Staubli VAL3: Vplus.dtx

jointRx jApproBox = {j4=-92.220275879, j3=-91.7603, j5=93.350395203, j1=-156.02204895, j2=-0.296387, j6=-204.139266968
}
jointRx jApproCam = {j4=-180, j3=-82.2022, j5=103.994537354, j1=17.642303467, j2=3.86292, j6=-29.504484177}
jointRx jApproConveyor = {j4=-180.000076294, j3=-104.09, j5=92.340240479, j1=-158.040847778, j2=16.4304, j6=-180.000152588}
jointRx jApproImm = {j4=-185.301483154, j3=-141.503, j5=-47.082424164, j1=105.804260254, j2=4.10028, j6=197.839569092}
jointRx jApproInspect = {j4=-180.122924805, j3=-94.165, j5=107.282814026, j1=79.97895813, j2=19.1074, j6=-27.049661636}
jointRx jApproReject = {j4=-180.000076294, j3=-82.9248, j5=105.547271729, j1=-36.019268036, j2=7.53623, j6=-53.689052582}
jointRx jApproSink = {j4=-180, j3=-82.9248, j5=105.547271729, j1=57.782627106, j2=7.53623, j6=-53.689052582}
jointRx jApproTurn = {j4=-180.000076294, j3=-91.6509, j5=105.937507629, j1=-68.973823547, j2=15.2445, j6=-24.155277252}
jointRx jApproWeld = {j4=-180, j3=-97.4879, j5=76.231643677, j1=-117.552749634, j2=-9.04277, j6=-203.299514771}
pointRx pCamCoords = {rx=0, x=143.13, ry=0, z=0, rz=-124.14, y=76.87, fatherId=world[0]}
pointRx pCamOrig = {rx=0.088055, x=-777.298, ry=177.401, z=14.3041, rz=-179.442, y=67.5964, fatherId=world[0]}
pointRx pCamX = {rx=0.0877556, x=-688.671, ry=177.399, z=15.1582, rz=-179.444, y=-158.575, fatherId=world[0]}
pointRx pCamY = {rx=0.0885309, x=-610.055, ry=177.399, z=12.4062, rz=-179.445, y=133.542, fatherId=world[0]}
tool pGripper0deg = {rx=0, x=0, ry=0, z=400, rz=0, ioLink=valve1, y=2, fatherId=flange[0]}
tool pGripper90deg = {rx=-89.9802, x=0, ry=0, z=312.5, rz=0, ioLink=valve1, y=-87.5, fatherId=flange[0]}
jointRx jHome = {j4=-180, j3=-104.09, j5=92.340240479, j1=-89.999916077, j2=16.4304, j6=-180.000152588}
pointRx pInspection = {rx=-0.828271, x=-402.297, ry=179.533, z=45.3187, rz=71.0887, y=-398.404, fatherId=world[0]}
pointRx pPickImm = {rx=-0.0335721, x=713.865, ry=88.1187, z=-110.012, rz=142.138, y=-1042.29, fatherId=world[0]}
pointRx pPickLoc = {rx=-0.45978, x=-648.514, ry=-179.559, z=13.9554, rz=-173.639, y=-37.8477, fatherId=world[0]}
pointRx pPickTurn = {rx=0.649757, x=-388.63, ry=179.139, z=10.1432, rz=-89.9458, y=350.625, fatherId=world[0]}
pointRx pPickWeld = {rx=-0.721699, x=-100.432, ry=-2.56053, z=-8.67817, rz=-71.824, y=700.057, fatherId=world[0]}
pointRx pPlaceBox[3]
  [0] = {rx=-0.00931083, x=744.888, ry=26.8991, z=177.661, rz=31.4855, y=890.517, fatherId=world[0]}
  [1] = {rx=-0.00931083, x=744.888, ry=26.8991, z=177.661, rz=31.4855, y=890.517, fatherId=world[0]}
  [2] = {rx=-0.00931083, x=744.888, ry=26.8991, z=177.661, rz=31.4855, y=890.517, fatherId=world[0]}
  [3] = {rx=-0.00931083, x=744.888, ry=26.8991, z=177.661, rz=31.4855, y=890.517, fatherId=world[0]}
pointRx pPlaceBoxRejec = {rx=-33.9923, x=393.165, ry=-30.0331, z=496.328, rz=22.9459, y=839.667, fatherId=world[0]}
pointRx pPlaceCover
  [0] = {rx=-3.39884, x=-140.67, ry=-2.89406, z=11.5788, rz=-72.075, y=727.524, fatherId=world[0]}
  [1] = {rx=4.46172, x=-55.7643, ry=-2.8981, z=-7.34839, rz=-72.4729, y=700.328, fatherId=world[0]}
pointRx pPlaceImm = {rx=2.40564, x=695.557, ry=88.1161, z=-100.844, rz=140.773, y=-867.761, fatherId=world[0]}
pointRx pPlaceReject = {rx=-0.758349, x=-362.79, ry=179.442, z=-135.753, rz=-101.683, y=177.761, fatherId=world[0]}
pointRx pPlaceSink = {rx=23.517, x=-427.516, ry=179.533, z=57.5011, rz=68.2962, y=-256.819, fatherId=world[0]}
pointRx pPlaceTurn = {rx=-2.72726, x=-533.365, ry=-4.55086, z=274.72, rz=-93.0403, y=527.16, fatherId=world[0]}
pointRx pPlaceWeld = {rx=-0.773504, x=38.7997, ry=178.381, z=-171.963, rz=108.632, y=668.081, fatherId=world[0]}
pointRx pPointer = {rx=0, x=0, ry=0, z=100, rz=0, y=0, fatherId=world[0]}
pointRx pRejectConveyor = {rx=33.9051, x=1007.54, ry=164.888, z=-263.078, rz=-97.3551, y=252.877, fatherId=world[0]}
pointRx pRob2Cam = {rx=0.604422, x=-777.298, ry=0.201455, z=14.3041, rz=68.6039, y=67.5964, fatherId=world[0]}
pointRx pWaitImm = {rx=2.56238, x=399.291, ry=88.3742, z=-104.522, rz=146.934, y=-634.763, fatherId=world[0]}
